// TIA Portal V17 export
// export: Created 2024-06-14T09:53:52.6814383Z, ExportSetting WithDefaults, DisplayName Totally Integrated Automation Portal, DisplayVersion V17, DisplayName TIA Portal Openness, DisplayVersion V17, DisplayName TIA Portal Version Control Interface, DisplayVersion V17, DisplayName Simotion SCOUT TIA, DisplayVersion 5.4.3.0, DisplayName SINAMICS Startdrive Advanced, DisplayVersion V17 SP1 Update 1, DisplayName SINAMICS Startdrive G110M, G120, G120C, G120D, G120P, G115D, DisplayVersion V17 SP1 Update 1, DisplayName SINAMICS Startdrive G130, G150, S120, S150, SINAMICS MV, S210, DisplayVersion V17 SP1 Update 1, DisplayName STEP 7 Professional, DisplayVersion V17, DisplayName STEP 7 Safety, DisplayVersion V17, DisplayName WinCC Professional, DisplayVersion V17
TYPE "Mod_Connect_Data"
// stored: IsFailsafeCompliant false
   STRUCT
      connectParamClient { S7_SetPoint := 'True'} : TCON_IP_v4;
   END_STRUCT;
   // connectParamClient.InterfaceId := 64;
   // connectParamClient.ID := 16#2;
   // connectParamClient.ActiveEstablished := true;
   // connectParamClient.RemoteAddress.ADDR[1] := 192;
   // connectParamClient.RemoteAddress.ADDR[2] := 168;
   // connectParamClient.RemoteAddress.ADDR[3] := 0;
   // connectParamClient.RemoteAddress.ADDR[4] := 3;
   // connectParamClient.RemotePort := 503;
   // connectParamClient.LocalPort := 0;
END_TYPE
